// TIA Portal V20 export
TYPE "LER_TypeFATMode_Capability_ProcessValue"
// stored: Access Published
   STRUCT
      CapabilityCount : Int;
      SelectCycle_ProcessValue : Int;
   END_STRUCT;
END_TYPE
